Staubli VAL3: N13_Ampolla.pgx

program N13_Ampolla()
  local pointRx l_pAmpolla
begin

  // Anar al punt de l'ampolla
  l_pAmpolla=pAmpolla[aioGet(aiNumAmpolla)]
  l_pAmpolla.trsf.x=l_pAmpolla.trsf.x+nXOffset
  l_pAmpolla.trsf.y=l_pAmpolla.trsf.y+nYOffset
  l_pAmpolla.trsf.z=l_pAmpolla.trsf.z+nZOffset
  movel(l_pAmpolla,tToolActiva,mLent)
  waitEndMove()

  bTaskDone=true
end
